TYPE TankCtrl_Priv :
STRUCT
	// State Manger
	smgr					: I_StateManager;
	
	// Flags
	IsSystemOn				: Flag;
	
	// Resources
	nErrorCode				: USINT;
	tankBuffer				: TagBuffer<CST.MAX_TANK>;
	
	iTank					: I_Domain;
	sTankId					: Str;
	
END_STRUCT
END_TYPE

(* stored: Version 1.1.0.1
   DUT TankCtrl_Priv: Id {9215b58a-206d-48c8-945c-7863e89017d6} *)
